if not RENDER:
    RDK.Render(False)

# Iterate through all joints in the matrix and check for collisions
njoints_all = jlist.size(1)
for i in range(njoints_all):
    ji = jlist[:,i].tolist()

    # Update the robot to a new position (it will create a new particle)
    robot.setJoints(ji)
    if not RENDER:
        # If Render is turned off (faster) update the position to draw a new particle
        RDK.Update()

    # Show a message in the RoboDK status bar from time to time
    if i % 10 == 0:
        msg = "Quick material deposition simulation for %s (%.1f %%)" % (progname, 100.0*(i/njoints_all))
        print(msg)
        RDK.ShowMessage(msg, False)

    # Render from time to time even if we have render deactivated
    if not RENDER and i % 500 == 0:
        RDK.Render()

RDK.Render(True)
msg = "Done"
print("Done")
RDK.ShowMessage(msg, False)
